Staubli VAL3: MsgType.dtx

public num PING
public num GET_VERSION
public num JOINT_POSITION
public num JOINT_TRAJ
public num JOINT_TRAJ_PT
public num JOINT_TRAJ_PT_F
public num JOINT_FEEDBACK
public num STATUS
